{attribute addProperty BoxType "ELX3351-0000-0016"}
{attribute addProperty Id "OverrangeBIT10.1252Data_invalidBIT10.1254ErrorBIT10.1257Calibration_in_progressBIT10.1258Steady_stateBIT10.1259TxPDO_ToggleBIT10.12516"}
{attribute addProperty CRC "3406431923"}
{attribute addProperty SizeInBites "16"}
{attribute addProperty SizeInBytes "2"}
TYPE Status_CB0A06B3 :
STRUCT
	{attribute 'hide'}
	reserve_1 : BIT;
	{attribute addProperty Name "Overrange"}
	Overrange : BIT;
	{attribute 'hide'}
	reserve_2 : BIT;
	{attribute addProperty Name "Data_invalid"}
	Data_invalid : BIT;
	{attribute 'hide'}
	reserve_3_BIT_0 : BIT;
	{attribute 'hide'}
	reserve_3_BIT_1 : BIT;
	{attribute addProperty Name "Error"}
	Error : BIT;
	{attribute addProperty Name "Calibration_in_progress"}
	Calibration_in_progress : BIT;
	{attribute addProperty Name "Steady_state"}
	Steady_state : BIT;
	{attribute 'hide'}
	reserve_4_BIT_0 : BIT;
	{attribute 'hide'}
	reserve_4_BIT_1 : BIT;
	{attribute 'hide'}
	reserve_4_BIT_2 : BIT;
	{attribute 'hide'}
	reserve_4_BIT_3 : BIT;
	{attribute 'hide'}
	reserve_4_BIT_4 : BIT;
	{attribute 'hide'}
	reserve_4_BIT_5 : BIT;
	{attribute addProperty Name "TxPDO_Toggle"}
	TxPDO_Toggle : BIT;
END_STRUCT
END_TYPE

(* stored: Version 1.2.0.0, ProductVersion 3.1.4024.9
   DUT Status_CB0A06B3: Id {1e99b0ad-983b-4323-9fe0-e0dac982d28c} *)
